FUNCTION_BLOCK SET_DEPTH (* Sets the final depth of a hole depending on its conditions *)
  (* Standard: 61499-2 *)
  (* Version 1.0, 09-01-12, Guilherme Jarentchuk, Universidade do Estado de Santa Catarina *)
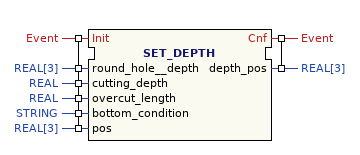
  EVENT_INPUT
    Init WITH round_hole__depth, cutting_depth, overcut_length, bottom_condition, pos; (* Initialize execution *)
  END_EVENT
  EVENT_OUTPUT
    Cnf WITH depth_pos; (* Confirm execution *)
  END_EVENT
  VAR_INPUT
    round_hole__depth : ARRAY [0..2] OF REAL; (* Coordinates of the plan that contains hole depth *)
    cutting_depth : REAL := 0; (* Overrides depth value and overcut *)
    overcut_length : REAL := 0; (* Amount of overcut *)
    bottom_condition : STRING; (* Types: "blind" or "through" *)
    pos : ARRAY [0..2] OF REAL; (* Machine position *)
  END_VAR
  VAR_OUTPUT
    depth_pos : ARRAY [0..2] OF REAL; (* Depth position *)
  END_VAR
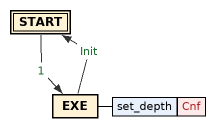
  EC_STATES
    START;
    EXE : set_depth -> Cnf;
  END_STATES
  EC_TRANSITIONS
    START TO EXE := 1;
    EXE TO START := Init;
  END_TRANSITIONS
  ALGORITHM set_depth IN Lua:
if ( cutting_depth > 0 ) then
	depth_pos[ 1 ] = pos[ 1 ]
	depth_pos[ 2 ] = pos[ 2 ]
	depth_pos[ 3 ] = pos[ 3 ] - cutting_depth
elseif( bottom_condition == 'BLIND_BOTTOM_CONDITION' ) then
	depth_pos[ 1 ] = pos[ 1 ]
	depth_pos[ 2 ] = pos[ 2 ]
	depth_pos[ 3 ] = pos[ 3 ] + round_hole__depth[ 3 ]
elseif( bottom_condition == 'THROUGH_BOTTOM_CONDITION' ) then
	depth_pos[ 1 ] = pos[ 1 ]
	depth_pos[ 2 ] = pos[ 2 ]
	depth_pos[ 3 ] = pos[ 3 ] + round_hole__depth[ 3 ] - overcut_length
end
  END_ALGORITHM
END_FUNCTION_BLOCK
